{attribute addProperty BoxType "IODEVICETYPE_ETHERCATPROT"}
{attribute addProperty Id "Beckhoff_ELXxxxxBeckhoff_ELXxxxx_091FCA884543567.875SyncUnitsSyncUnits_CAB22D3B19524.375InputsInputs_C75D3FEC1280160OutputsOutputs_47D1E803848106InfoDataInfoData_E9F65A829612"}
{attribute addProperty CRC "58353333"}
{attribute addProperty SizeInBites "6962"}
{attribute addProperty SizeInBytes "870.25"}
TYPE EtherCAT_Master_ELXxxxx_037A66B5 :
STRUCT
	{attribute addProperty Name "Beckhoff_ELXxxxx"}
	Beckhoff_ELXxxxx : Beckhoff_ELXxxxx_091FCA88;
	{attribute addProperty Name "SyncUnits"}
	SyncUnits : SyncUnits_CAB22D3B;
	{attribute addProperty Name "Inputs"}
	Inputs : Inputs_C75D3FEC;
	{attribute addProperty Name "Outputs"}
	Outputs : Outputs_47D1E803;
	{attribute addProperty Name "InfoData"}
	InfoData : InfoData_E9F65A82;
END_STRUCT
END_TYPE

(* stored: Version 1.2.0.0, ProductVersion 3.1.4024.9
   DUT EtherCAT_Master_ELXxxxx_037A66B5: Id {4066de18-9c7d-41fa-9eeb-b083ca757bab} *)
